FUNCTION F_ITC_SendTDR : BOOL
(**************************************************************************************
 * 	Application		:	BoxControl Framework
 *	Revision		:	$Revision: 404529 $
 *	Revision date	:	$Date: 2018-04-23 08:21:38 +0200 (Mo., 23 Apr 2018) $
 *	Last changed by	:	$Author: b7bolm $
 *	URL				:	$URL: http://almscdc.swisslog.com/repo/SWPD/Development/BoxControlFramework/20_Release/trunk/01_Software/BCF/BCF/JumpStart/20_Product/10_App/11_Com/10_Lib/10_Conv/11_ITC/F_ITC_SendTDR.TcPOU $
 *
 *	Purpose			:	Wrap message - TDR
 *
 * ------------------------------------------------------------------------------------
 *	Copyright Swisslog [IP AG], Switzerland. All rights reserved.
 * 
 * ------------------------------------------------------------------------------------
 *	
 * 	Revision History: 
 *
 * 	VERSION			DATE			INITIALS			DESCRIPTION
 *	0.1				01.01.2001		swl					Example
 *
 **************************************************************************************)
VAR_INPUT
	eChannelSrc		: E_MFCS_Channel; // Source communicaton channel	
	PositionName	: STRING(Conveyor.POSITION_STRINGLENGTH); // SIS MM-GGG-EEEE-FF-Z
	TU_ID			: STRING(Conveyor.TU_ID_STRINGLENGTH); // 18 Digit SSID
	AssignmentID	: UDINT; // assignment id
	MsgSequence		: INT; // MSG Sequence
	eReturnCode		: E_ErrorConv; // Return code
END_VAR
VAR
	TDR				: ST_ITC_TDR; 
END_VAR

// Map values
TDR.Position := PositionName;
TDR.TU_ID := TU_ID;
TDR.AssignmentID := AssignmentID;
TDR.MsgSequence := MsgSequence;
TDR.ReturnCode := eReturnCode;

// Forward to ITC
F_ITC_SendTDR := fbITC_Manager.M_SendData(
					meChannel	:= eChannelSrc,
					mMsgType	:= E_ITC_MsgTypeConv.TASK_DELETE_REPORT,
					mpData		:= ADR(TDR),
					mLen		:= SIZEOF(TDR));

END_FUNCTION

(* stored: Version 1.1.0.1, ProductVersion 3.1.4022.12
   POU F_ITC_SendTDR: Id {f266fab2-7915-4e26-a17c-ef2c19f9d000}, SpecialFunc None *)
